FUNCTION_BLOCK FB_RecipeBuilderBorgoFlaps EXTENDS FB_RecipeBase

METHOD Build : BOOL
VAR_INST
    TotalY          : REAL;
    TotalX          : REAL;
    ShorterY        : REAL;
    ShorterX        : REAL;
END_VAR
_Busy := TRUE;
_Done := FALSE;
_Error := FALSE;
Build := FALSE;

THIS^.UpdateNestingLimits();

// 2. Jeśli detal wystaje poza maszynę - przerywamy od razu!
IF NOT _Config.IsValid THEN
    _Busy := FALSE;
    _Error := TRUE; 
    Build := FALSE;
    RETURN;
END_IF

// 3. Pobieramy wyliczone gabaryty nominalne do lokalnych zmiennych roboczych
TotalX   := _NominalX;
TotalY   := _NominalY; 
ShorterY := TotalY - _Config.PanelHeight;
ShorterX := TotalX - _Config.PanelHeight;


// ------------------------------------
// 1. Segregracja frezowania (Grooving)
// ------------------------------------
_SegmentsToGroove := 4;

_SegmentsGroove[1].Start.X := TotalX;
_SegmentsGroove[1].Stop.X  := 0;
_SegmentsGroove[1].Start.Y := ShorterY;
_SegmentsGroove[1].Stop.Y  := ShorterY;

_SegmentsGroove[2].Start.X := TotalX;
_SegmentsGroove[2].Stop.X  := 0; 
_SegmentsGroove[2].Start.Y := _Config.PanelHeight;
_SegmentsGroove[2].Stop.Y  := _Config.PanelHeight;

_SegmentsGroove[3].Start.X := ShorterX;
_SegmentsGroove[3].Stop.X  := ShorterX;
_SegmentsGroove[3].Start.Y := TotalY;
_SegmentsGroove[3].Stop.Y  := 0;

_SegmentsGroove[4].Start.Y := TotalY;
_SegmentsGroove[4].Stop.Y  := 0;
_SegmentsGroove[4].Start.X := _Config.PanelHeight;
_SegmentsGroove[4].Stop.X  := _Config.PanelHeight;

// ------------------------------------
// 2. Cięcie w osi X (Cut X)
// ------------------------------------
_SegmentsToCutX := 6;

// Short Box Segments
_SegmentsCutX[1].Start.X := TotalX + _Config.CuttingOverpass;
_SegmentsCutX[1].Stop.X  := ShorterX;
_SegmentsCutX[1].Start.Y := ShorterY;
_SegmentsCutX[1].Stop.Y  := ShorterY;

_SegmentsCutX[2].Start.X := _Config.PanelHeight;
_SegmentsCutX[2].Stop.X  := -_Config.CuttingOverpass;
_SegmentsCutX[2].Start.Y := ShorterY;
_SegmentsCutX[2].Stop.Y  := ShorterY;

_SegmentsCutX[3].Start.X := TotalX + _Config.CuttingOverpass;
_SegmentsCutX[3].Stop.X  := ShorterX;
_SegmentsCutX[3].Start.Y := _Config.PanelHeight;
_SegmentsCutX[3].Stop.Y  := _Config.PanelHeight;

_SegmentsCutX[4].Start.X := _Config.PanelHeight;
_SegmentsCutX[4].Stop.X  := -_Config.CuttingOverpass;
_SegmentsCutX[4].Start.Y := _Config.PanelHeight;
_SegmentsCutX[4].Stop.Y  := _Config.PanelHeight;

// Panel Dimensions 
_SegmentsCutX[5].Start.X := TotalX + _Config.CuttingOverpass;
_SegmentsCutX[5].Stop.X  := -_Config.CuttingOverpass;
_SegmentsCutX[5].Start.Y := TotalY;
_SegmentsCutX[5].Stop.Y  := TotalY;

_SegmentsCutX[6].Start.X := TotalX + _Config.CuttingOverpass;
_SegmentsCutX[6].Stop.X  := -_Config.CuttingOverpass;
_SegmentsCutX[6].Start.Y := 0;
_SegmentsCutX[6].Stop.Y  := 0;

// ------------------------------------
// 3. Cięcie w osi Y (Cut Y)
// ------------------------------------
_SegmentsToCutY := 6;

// Short Box Segments
_SegmentsCutY[1].Start.X := ShorterX;
_SegmentsCutY[1].Stop.X  := ShorterX;
_SegmentsCutY[1].Start.Y := TotalY + _Config.CuttingOverpass;
_SegmentsCutY[1].Stop.Y  := ShorterY;

_SegmentsCutY[2].Start.X := _Config.PanelHeight;
_SegmentsCutY[2].Stop.X  := _Config.PanelHeight;
_SegmentsCutY[2].Start.Y := TotalY + _Config.CuttingOverpass;
_SegmentsCutY[2].Stop.Y  := ShorterY;

_SegmentsCutY[3].Start.X := ShorterX;
_SegmentsCutY[3].Stop.X  := ShorterX;
_SegmentsCutY[3].Start.Y := _Config.PanelHeight;
_SegmentsCutY[3].Stop.Y  := -_Config.CuttingOverpass;

_SegmentsCutY[4].Start.X := _Config.PanelHeight;
_SegmentsCutY[4].Stop.X  := _Config.PanelHeight;
_SegmentsCutY[4].Start.Y := _Config.PanelHeight;
_SegmentsCutY[4].Stop.Y  := -_Config.CuttingOverpass;

// Panel Dimensions Shorter Wings
_SegmentsCutY[5].Start.X := TotalX - _Config.RailHeightCorrection;
_SegmentsCutY[5].Stop.X  := TotalX - _Config.RailHeightCorrection;
_SegmentsCutY[5].Start.Y := TotalY + _Config.CuttingOverpass;
_SegmentsCutY[5].Stop.Y  := -_Config.CuttingOverpass;

_SegmentsCutY[6].Start.X := _Config.RailHeightCorrection;
_SegmentsCutY[6].Stop.X  := _Config.RailHeightCorrection;
_SegmentsCutY[6].Start.Y := TotalY + _Config.CuttingOverpass;
_SegmentsCutY[6].Stop.Y  := -_Config.CuttingOverpass;


_Busy := FALSE;
_Done := TRUE;
Build := TRUE;
END_METHOD

METHOD PROTECTED CalculateFootprint
VAR_INPUT
END_VAR
// BorgoWings wie, że jego wymiar powiększa się o ścianki zagięcia:
_NominalX := _Config.PanelFrontWidth  + 2.0 * _Config.PanelHeight; 
_NominalY := _Config.PanelFrontLength + 2.0 * _Config.PanelHeight;
END_METHOD

PROPERTY ExecutionRoute : E_ExecutionRoute
GET
ExecutionRoute := E_ExecutionRoute.ePTP;
END_GET
END_PROPERTY

METHOD FB_init : BOOL
VAR_INPUT
	bInitRetains : BOOL; // if TRUE, the retain variables are initialized (warm start / cold start)
	bInCopyCode : BOOL;  // if TRUE, the instance afterwards gets moved into the copy code (online change)
END_VAR
_Limits.PanelFrontLength.MinVal := 100.0;
_Limits.PanelFrontLength.MaxVal := 2400.0;

_Limits.PanelFrontWidth.MinVal  := 100.0;
_Limits.PanelFrontWidth.MaxVal  := 1200.0;

_Limits.PanelHeight.MinVal      := 40.0;
_Limits.PanelHeight.MaxVal      := 100.0;

_Limits.RailHeightCorrection.MinVal := 12.0;
_Limits.RailHeightCorrection.MaxVal := 14.0;

_Limits.CuttingOverpass.MinVal := 0.0;
_Limits.CuttingOverpass.MaxVal := 50.0;

_Limits.GroovingOverpass.MinVal := 0.0;
_Limits.GroovingOverpass.MaxVal := 50.0;

_Limits.GrooveDepthZ.MinVal := 0.0;
_Limits.GrooveDepthZ.MaxVal := 9.0; //
END_METHOD

END_FUNCTION_BLOCK

(* stored: Version 1.1.0.1, ProductVersion 3.1.4024.15
   POU FB_RecipeBuilderBorgoFlaps: Id {1389b747-8c88-4122-8f76-112cbf46c424}, SpecialFunc None
   Method Build: Id {a7636aac-6540-4877-9111-d7366342a8fe}
   Method CalculateFootprint: Id {9729302b-8841-4a61-a0ae-d9106fc641a1}
   Property ExecutionRoute: Id {0305d75c-974a-4eab-a51e-af357ba6ad95}
   Get Get: Id {656fd98a-8440-4295-ade6-b1b129d2e1b8}
   Method FB_init: Id {4a0331ae-cce1-43c4-8f3f-519ce38c4c04} *)
